FUNCTION_BLOCK INTERNAL FINAL FB_RoundTripRepeatedFieldStringTests EXTENDS FB_TestSuite
VAR CONSTANT
    cExpected 			: ARRAY[0..7] OF STRING := ['abc', '123', '🤖👾�', 'ABCDEFG HIJK', 'äöüß'];
	cExpectedFieldIndex : UDINT := 5;
END_VAR
VAR
    aBuffer         	: ARRAY[0..255] OF BYTE;
    hrWriterActual  	: HRESULT;
    hrParserActual  	: HRESULT;
	aActuals, aValues	: ARRAY[0..7] OF STRING ;
	nActualTag			: UDINT;
	nExpectedTag	    : UDINT;
    fbParseCtx_SUT      : FB_ParseContext;
	fbWriteCtx_SUT		: FB_WriteContext;
	fbFieldCodec 		: FB_FieldCodecString(nTag:= F_MakeTag(nFieldNumber:= 3, eWireType:= E_WireType.LengthDelimited));
	fbRepeatedField_Write : FB_RepeatedField(anyArray:= F_ToAnyType(aValues), anyFirstElem:= F_ToAnyType(aValues[0]), ipFieldCodec:= fbFieldCodec);
	fbRepeatedField_Parse : FB_RepeatedField(anyArray:= F_ToAnyType(aActuals), anyFirstElem:= F_ToAnyType(aActuals[0]), ipFieldCodec:= fbFieldCodec);
END_VAR
VAR_TEMP
	i : INT;
END_VAR

TEST(__POUNAME());

// Arrange
nExpectedTag := F_MakeTag(nFieldNumber:= 3, eWireType:= E_WireType.LengthDelimited);
aValues := cExpected;
fbRepeatedField_Write.InitializeFromArray(anyArray:= F_ToAnyType(aValues), anyFirstElem:= F_ToAnyType(aValues[0]), nCount:= 5);
fbWriteCtx_SUT.FromBuffer(aBuffer);
fbParseCtx_SUT.FromBuffer(aBuffer);

// Act

hrWriterActual := fbRepeatedField_Write.WriteTo(fbWriteCtx_SUT, fbFieldCodec);
fbParseCtx_SUT.ReadTag(nTag=> nActualTag);
hrParserActual := fbRepeatedField_Parse.AddEntriesFrom(fbParseCtx_SUT, fbFieldCodec);

// Assert

AssertEquals_DINT(Expected:= S_OK, Actual:= hrWriterActual, Message:= 'Expected hrWriterActual = S_OK');
AssertEquals_DINT(Expected:= S_OK, Actual:= hrParserActual, Message:= 'Expected hrParserActual = S_OK');
AssertEquals_UDINT(Expected:= nExpectedTag, Actual:= nActualTag, Message:= 'Expeced nActualTag to equal nExpectedTag.');
AssertEquals_UDINT(Expected:= cExpectedFieldIndex, Actual:= fbRepeatedField_Parse.nCount, Message:= 'Expeced fbRepeatedField_Parse.nCount to equal cExpectedFieldIndex.');

FOR i := 0 TO 7 DO 
	AssertEquals_STRING(Expected:= cExpected[i], Actual:= aActuals[i], Message:= CONCAT(CONCAT('Index ', TO_STRING(i)), ' differ'));
END_FOR

TEST_FINISHED_NAMED(__POUNAME());

END_FUNCTION_BLOCK

(* stored: Version 1.1.0.1
   POU FB_RoundTripRepeatedFieldStringTests: Id {ef15ae40-4d23-48db-af8c-71c9ce8a70f7}, SpecialFunc None *)
